FUNCTION_BLOCK fbRealToDWord
VAR_INPUT
	in_r_Value				: REAL ;
	in_r_Res				: REAL ;
	in_i_Offset				: INT ;
END_VAR
VAR_OUTPUT
	out_B0					: BYTE ;
	out_B1					: BYTE ;
	out_B2					: BYTE ;
	out_B3					: BYTE ;
END_VAR
VAR
	dw_AddedValue			: DWORD;
	r_ResolutionResolved	: REAL;
	r_OffsetSolved			: REAL;
END_VAR

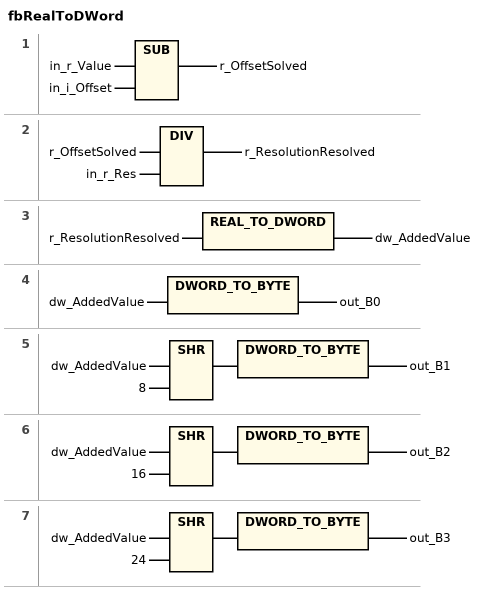
// NETWORK 1
r_OffsetSolved := in_r_Value - in_i_Offset;

// NETWORK 2
r_ResolutionResolved := r_OffsetSolved / in_r_Res;

// NETWORK 3
dw_AddedValue := REAL_TO_DWORD(r_ResolutionResolved);

// NETWORK 4
out_B0 := DWORD_TO_BYTE(dw_AddedValue);

// NETWORK 5
out_B1 := DWORD_TO_BYTE(SHR(dw_AddedValue, 8));

// NETWORK 6
out_B2 := DWORD_TO_BYTE(SHR(dw_AddedValue, 16));

// NETWORK 7
out_B3 := DWORD_TO_BYTE(SHR(dw_AddedValue, 24));

END_FUNCTION_BLOCK

(* stored: Version 1.1.0.1, ProductVersion 3.1.4024.12
   POU fbRealToDWord: Id {c067c25f-45ea-44b8-8bf3-818176233c42}, SpecialFunc None *)
